FUNCTION_BLOCK FB_Invoke
VAR_INPUT
END_VAR
VAR_OUTPUT
END_VAR
VAR
END_VAR

END_FUNCTION_BLOCK

(* stored: Version 1.1.0.1, ProductVersion 3.1.4022.12
   POU FB_Invoke: Id {41eb7c5d-132f-4e51-bd5c-da9f681236c9}, SpecialFunc None *)
